FUNCTION_BLOCK SORTER_SAMPLE_COLOR (* Composite Function Block Type *)
  (* Standard: 61499-2 *)
  (* Version 0.0, 1/27/2023, brink, Flexbridge AB, template *)
  PACKAGE UAO.Hackathon;
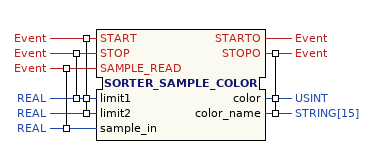
  EVENT_INPUT
    START WITH limit1, limit2; (* Start detection *)
    STOP WITH limit1; (* Stop detecton and save detected values *)
    SAMPLE_READ WITH sample_in;
  END_EVENT
  EVENT_OUTPUT
    STARTO; (* Detection started *)
    STOPO WITH color, color_name; (* Detection stopped *)
  END_EVENT
  VAR_INPUT
    limit1 : REAL;
    limit2 : REAL;
    sample_in : REAL; (* Input value from analog sensor *)
  END_VAR
  VAR_OUTPUT
    color : USINT;
    color_name : STRING[15];
  END_VAR
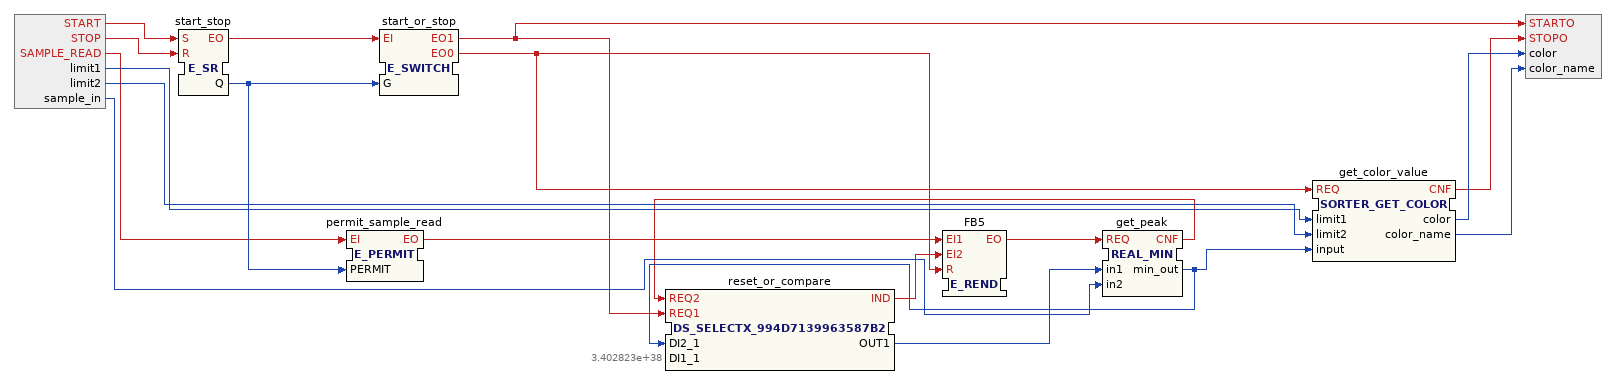
  FBS
    start_stop : E_SR;
    permit_sample_read : E_PERMIT;
    get_peak : REAL_MIN;
    get_color_value : SORTER_GET_COLOR;
    start_or_stop : E_SWITCH;
    reset_or_compare : DS_SELECTX_994D7139963587B2(DI1_1 := 3.402823e+38); {SET_ATTRIBUTE(Configuration.GenericFBType.InterfaceParams, Runtime.Standard#CNTX:=2;CNTY:=1;DI${CNTX,_,CNTY$}:REAL)}
    FB5 : E_REND;
  END_FBS
  EVENT_CONNECTIONS
    SAMPLE_READ TO permit_sample_read.EI;
    get_peak.CNF TO reset_or_compare.REQ2;
    permit_sample_read.EO TO FB5.EI1;
    FB5.EO TO get_peak.REQ;
    reset_or_compare.IND TO FB5.EI2;
    start_stop.EO TO start_or_stop.EI;
    start_or_stop.EO1 TO STARTO;
    start_or_stop.EO1 TO reset_or_compare.REQ1;
    start_or_stop.EO0 TO FB5.R;
    start_or_stop.EO0 TO get_color_value.REQ;
    get_color_value.CNF TO STOPO;
    START TO start_stop.S;
    STOP TO start_stop.R;
  END_CONNECTIONS
  DATA_CONNECTIONS
    get_color_value.color_name TO color_name;
    get_color_value.color TO color;
    limit1 TO get_color_value.limit1;
    limit2 TO get_color_value.limit2;
    get_peak.min_out TO get_color_value.input;
    start_stop.Q TO start_or_stop.G;
    get_peak.min_out TO reset_or_compare.DI2_1;
    reset_or_compare.OUT1 TO get_peak.in1;
    sample_in TO get_peak.in2;
    start_stop.Q TO permit_sample_read.PERMIT;
  END_CONNECTIONS
END_FUNCTION_BLOCK
